FUNCTION_BLOCK MotorCtrl (* Template for an empty basic function block *)
  (* Standard: 61499-2 *)
  (* Version 1.0, 2018-07-17, az *)
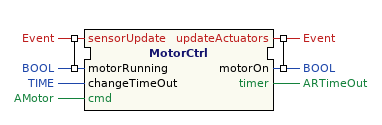
  EVENT_INPUT
    sensorUpdate WITH motorRunning;
  END_EVENT
  EVENT_OUTPUT
    updateActuators WITH motorOn;
  END_EVENT
  VAR_INPUT
    motorRunning : BOOL;
    changeTimeOut : TIME; (* time till the motor has either start moving or stopped moving after the according command was given *)
  END_VAR
  VAR_OUTPUT
    motorOn : BOOL;
  END_VAR
  SOCKETS
    cmd : AMotor;
  END_SOCKETS
  PLUGS
    timer : ARTimeOut;
  END_PLUGS
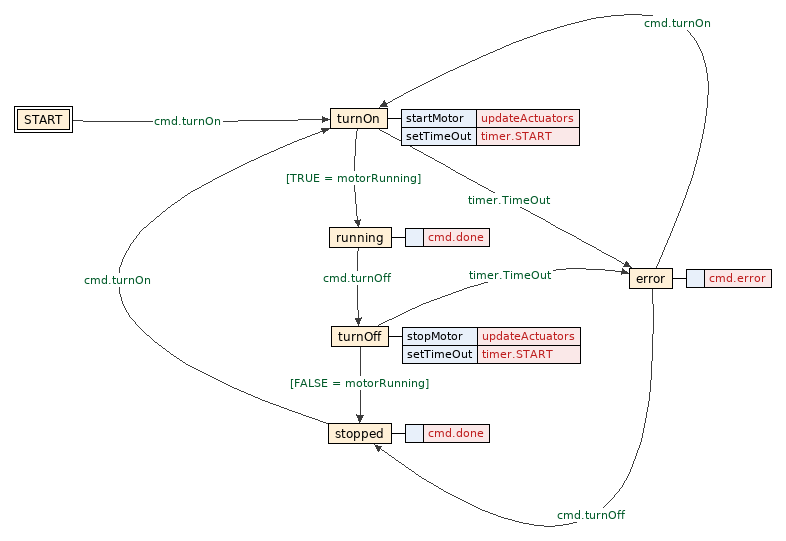
  EC_STATES
    START; (* Initial State *)
    turnOn : startMotor -> updateActuators, setTimeOut -> timer.START;
    running : -> cmd.done;
    turnOff : stopMotor -> updateActuators, setTimeOut -> timer.START;
    stopped : -> cmd.done;
    error : -> cmd.error;
  END_STATES
  EC_TRANSITIONS
    START TO turnOn := cmd.turnOn;
    turnOn TO running := [TRUE = motorRunning];
    running TO turnOff := cmd.turnOff;
    turnOff TO stopped := [FALSE = motorRunning];
    stopped TO turnOn := cmd.turnOn;
    turnOn TO error := timer.TimeOut;
    turnOff TO error := timer.TimeOut;
    error TO turnOn := cmd.turnOn;
    error TO stopped := cmd.turnOff;
  END_TRANSITIONS
  ALGORITHM startMotor IN ST: (* new algorithm *)
motorOn := TRUE;
  END_ALGORITHM
  ALGORITHM stopMotor IN ST: (* new algorithm *)
motorOn := FALSE;
  END_ALGORITHM
  ALGORITHM setTimeOut IN ST: (* new algorithm *)
timer.DT := changeTimeOut;
  END_ALGORITHM
END_FUNCTION_BLOCK
